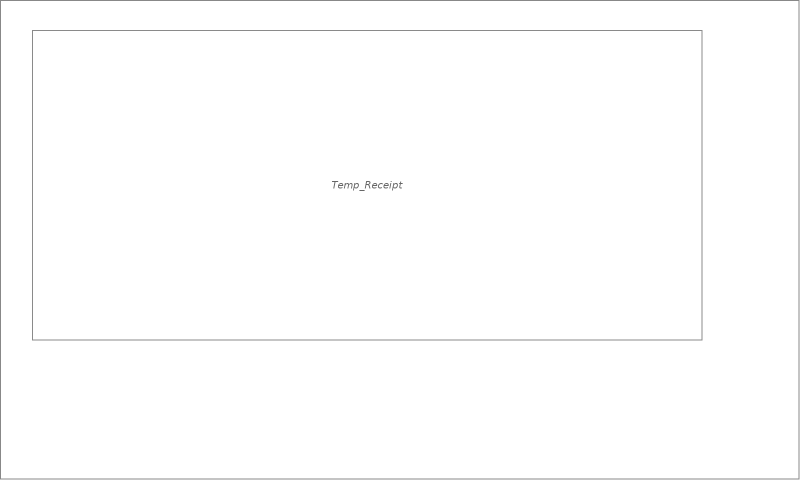
VISUALIZATION Visu_ReceiptList_02  // 800x480
    Frame (32,30 670x310)
        shows Temp_Receipt(stHmiRData := stRData[2])
END_VISUALIZATION

(* stored: Version 1.1.0.1, ProductVersion 3.1.4024.6
   Visu Visu_ReceiptList_02: Id {4f373a86-0877-487d-9b14-e86d179a7174} *)
